INTERFACE I_Stack EXTENDS I_Collections

(* Get item from stack without removing it. *)
METHOD Peek : I_Stack
VAR_INPUT
	Item 	: ANY; (* Variable to store returned item value *)
	nIndex 	: DINT; (* Location of item*)
END_VAR
END_METHOD

(* Gets and deletes item at the top of the stack *)
METHOD Pop : I_Stack
VAR_INPUT
	Item : ANY; (* Variable to store returned item value *)
END_VAR
END_METHOD

(* Removes item at the top of the stack without returning anything *)
METHOD Pop_Void : I_Stack
VAR_INPUT
END_VAR
END_METHOD

(* Add item to the top of the stack *)
METHOD Push : I_Stack
VAR_INPUT
	Item : ANY; (* Variable containg data to store on the stack *)
END_VAR
END_METHOD

(* Get item at the top of the stack without removing it. *)
METHOD Top : I_Stack
VAR_INPUT
	Item 	: ANY; (* Variable to store returned item value *)
END_VAR
END_METHOD

END_INTERFACE

(* stored: Version 1.1.0.1, ProductVersion 3.1.4024.4
   Itf I_Stack: Id {2df439e0-81da-4e78-87bf-c4adedd54744}
   Method Peek: Id {9a978ae2-f74e-4a80-a688-5ff02915b184}
   Method Pop: Id {3bcc8ffd-0585-4d63-8b9b-010f602fe127}
   Method Pop_Void: Id {48ea49e8-fe7d-43cc-92e3-4e500d8fe13c}
   Method Push: Id {80e4c8db-67e1-4c76-bcdb-e77d10437f1a}
   Method Top: Id {90510f03-ae76-443f-90c7-d276be0836b6} *)
